ABB RobotStudio station: 1200_station.rsstn

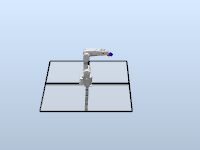
Station Station (saved by RobotStudio 21.4.9700.0)
Layout (positions relative to the parent item):
  - IRB1200_5_90_STD_03 [mechanism, from Robots\IRB1200_5_90_STD_03.rslib] at (0, 0, 0) mm; joint values [0, 0, 0, 0, 0.5236, 0] (rad or m)
